// TIA Portal V18 export
FUNCTION_BLOCK "select_remoteMP_FB"   // FB60, LAD
{ S7_Optimized_Access := 'TRUE' }
VERSION : 0.1
// stored: AutoNumber true, IsIECCheckEnabled false, IsRetainMemResEnabled false, MemoryReserve 100, SetENOAutomatically false, UDAEnableTagReadback false
   VAR_INPUT
      MD_AUtO : Bool;
      MD_DESK { ExternalAccessible := 'False'; ExternalVisible := 'False'; ExternalWritable := 'False'} : Bool;
      MD_RC { ExternalAccessible := 'False'; ExternalVisible := 'False'; ExternalWritable := 'False'} : Bool;
      Joystick { ExternalAccessible := 'False'; ExternalVisible := 'False'; ExternalWritable := 'False'} : Real;
      speed_RCfast { ExternalAccessible := 'False'; ExternalVisible := 'False'; ExternalWritable := 'False'} : Real;
   END_VAR
   VAR_OUTPUT
      speed { ExternalAccessible := 'False'; ExternalVisible := 'False'; ExternalWritable := 'False'} : Real;
   END_VAR
   VAR_IN_OUT
      m_AUTO : Bool;
      m_MAN : Bool;
   END_VAR
   VAR_TEMP
      slow_speed_static : Real;
      fast_speed_static : Real;
   END_VAR
BEGIN

REGION Network 1
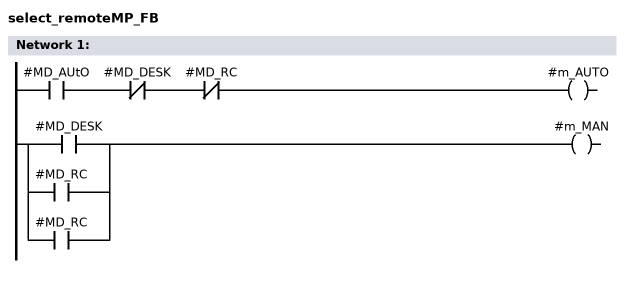
   RUNG wire#powerrail
      Contact( #MD_AUtO )
      I_Contact( #MD_DESK )
      I_Contact( #MD_RC )
      Coil( #m_AUTO )
   END_RUNG
   RUNG wire#powerrail
      Contact( #MD_DESK )
      wire#w1
      Coil( #m_MAN )
   END_RUNG
   RUNG wire#powerrail
      Contact( #MD_RC )
   END_RUNG wire#w1
   RUNG wire#powerrail
      Contact( #MD_RC )
   END_RUNG wire#w1
   // the same network as SCL:
   #m_AUTO := #MD_AUtO AND NOT #MD_DESK AND NOT #MD_RC;
   #m_MAN := #MD_DESK OR #MD_RC OR #MD_RC;
END_REGION
END_FUNCTION_BLOCK
